(* PLC project first_project, Beremiz beremiz 1 *)
(* stored: creationDateTime 2020-04-03T09:24:04, productRelease 1.0.0, modificationDateTime 2020-04-18T13:31:47, version 1.0.1 *)

(* 샘플 *)
PROGRAM program0
  VAR_INPUT
    p0001 : INT;
  END_VAR
  VAR_OUTPUT
    p0020 : INT;
  END_VAR
  VAR_TEMP
    p0003 : INT;
  END_VAR
  VAR_INPUT
    sw5 : INT;
  END_VAR
  VAR_OUTPUT
    led5 : INT;
  END_VAR

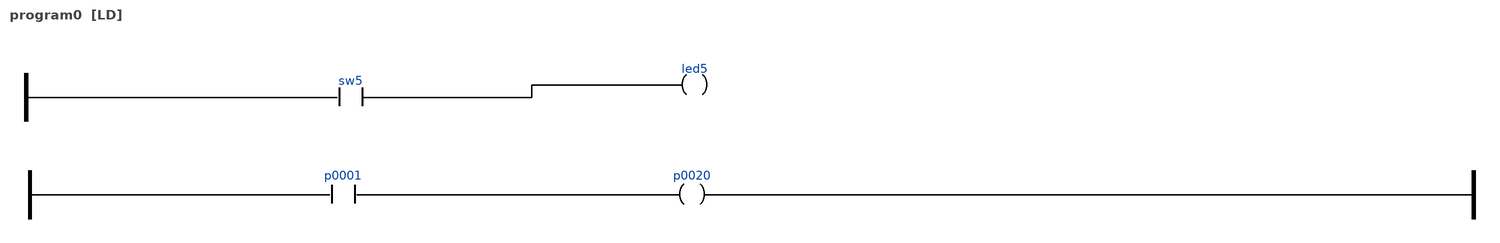
(* LD diagram, written out as Structured Text *)
led5 := sw5;
p0020 := p0001;
END_PROGRAM

CONFIGURATION config
  VAR_GLOBAL
    var1 : INT;
  END_VAR
  RESOURCE resource1 ON PLC
    TASK task0(INTERVAL := T#50ms, PRIORITY := 0);
    PROGRAM instance0 WITH task0 : program0;
  END_RESOURCE
END_CONFIGURATION
